(* IEC 61131-3 sources: my_OpenPLC_Editor/editor/arduino/src, 1 file *)

(* ---- plc_prog.st ---- *)
PROGRAM Blink
  VAR
    blink_led AT %QX0.3 : BOOL;
  END_VAR
  VAR
    TON0 : TON;
    TOF0 : TOF;
  END_VAR

  TON0(EN := TRUE, IN := NOT(blink_led), PT := T#500ms);
  TOF0(EN := TON0.ENO, IN := TON0.Q, PT := T#500ms);
  blink_led := TOF0.Q;
END_PROGRAM

CONFIGURATION Config0

  RESOURCE Res0 ON PLC
    TASK task0(INTERVAL := T#20ms,PRIORITY := 0);
    PROGRAM instance0 WITH task0 : Blink;
  END_RESOURCE
END_CONFIGURATION
